// Mitsubishi GX Works2 project: 231003-002- exercicios   PLC: Q03UDV

// global labels: Global1
VAR_GLOBAL
  Up_Down AT M34 : BOOL;
END_VAR

// task Task_01 (event TRUE, interval 0, priority 31): POU_01

PROGRAM POU_01
VAR
  CTD_1 : CTD;
  CTU_1 : CTU;
  meuc : CTU;
  novo : CTUD;
  TP_1 : TP;
  TON_1 : TON;
  TOF_1 : TOF;
  dr : TIME;
  timetp : TIME;
  timeon : TIME;
  TimeOFF : TIME;
  Input : BOOL;
  red : BOOL;
  TP_2 : TP;
  ver : BOOL;
  verd : BOOL;
  TP_3 : TP;
  amar : BOOL;
  Result : DINT;
END_VAR
(* structured ladder/FBD written out as ST: instructions are called as NAME(EN, inputs, outputs); _pN, _eN, _tN stand for wires *)
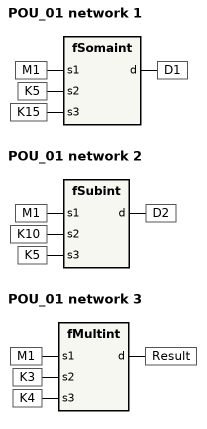
(* network 1 *)
D1 := fSomaint(M1, K5, K15);
(* network 2 *)
D2 := fSubint(M1, K10, K5);
(* network 3 *)
Result := fMultint(M1, K3, K4);
END_PROGRAM

FUNCTION fSomaint
VAR_INPUT
  i_xHabilitar : BOOL;
  i_iElemento1 : INT;
  i_iElemento2 : INT;
END_VAR
(* structured ladder/FBD written out as ST: instructions are called as NAME(EN, inputs, outputs); _pN, _eN, _tN stand for wires *)
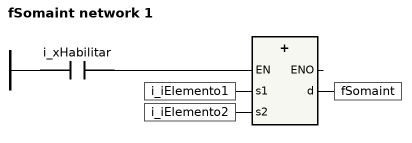
(* network 1 *)
+(i_xHabilitar, i_iElemento1, i_iElemento2, fSomaint);
END_FUNCTION

FUNCTION fSubint
VAR_INPUT
  i_xHabilitar : BOOL;
  i_iElemento1 : INT;
  i_iElemento2 : INT;
END_VAR
(* structured ladder/FBD written out as ST: instructions are called as NAME(EN, inputs, outputs); _pN, _eN, _tN stand for wires *)
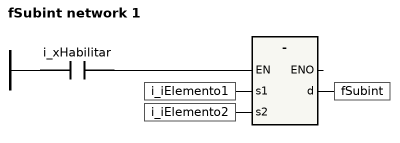
(* network 1 *)
-(i_xHabilitar, i_iElemento1, i_iElemento2, fSubint);
END_FUNCTION

FUNCTION fMultint  // d3
VAR_INPUT
  i_xHabilitar : BOOL;
  i_iElemento1 : INT;
  i_iElemento2 : INT;
END_VAR
(* structured ladder/FBD written out as ST: instructions are called as NAME(EN, inputs, outputs); _pN, _eN, _tN stand for wires *)
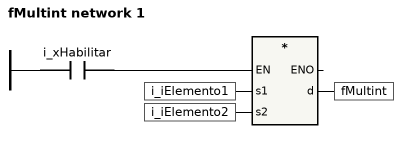
(* network 1 *)
*(i_xHabilitar, i_iElemento1, i_iElemento2, fMultint);
END_FUNCTION

FUNCTION fDivsaoint
(* structured ladder/FBD written out as ST: instructions are called as NAME(EN, inputs, outputs); _pN, _eN, _tN stand for wires *)
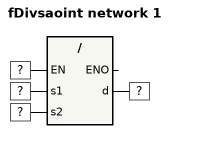
(* network 1 *)
/(?, ?, ?, ?);
END_FUNCTION
